// TwinCAT 3 PLC project H2AssemblyTesting
// ProgramVersion: 3.1.4026.17
// libraries:
//   Tc2_Standard, * (Beckhoff Automation GmbH)
//   Tc2_System, * (Beckhoff Automation GmbH)
//   Tc2_Utilities, * (Beckhoff Automation GmbH)
// project tree:
//   DUTs/ E_CompressionStages.TcDUT, E_ErrorState.TcDUT (not stored), E_InletToSystem.TcDUT (not stored), E_OutletNumber.TcDUT (not stored), E_TankBundleNumber.TcDUT (not stored), E_SolenoidState.TcDUT (not stored), ST_AnalogPressureTemp.TcDUT, ST_MatrixInputs.TcDUT, ST_Path.TcDUT (not stored), ST_SolenoidConfig.TcDUT
//   GVLs/ GVL_HMI.TcGVL, GVL_IO.TcGVL
//   / PlcTask.TcTTO (not stored)
//   POUs/ FB_Device.TcPOU, FB_IO.TcPOU, FB_Matrix.TcPOU, FB_PressureTransducer.TcPOU, FB_Solenoid.TcPOU, MAIN.TcPOU
//   POUs/Interfaces/ I_Devices.TcIO
// real-time tasks:
//   TASK PlcTask: cycle T#10ms, priority 20, ADS port 350
// I/O:
//   DEVICE Node 05 (disabled), AmsNetId 192.168.1.166.2.1
//     Node 05S0 [EK1100 EtherCAT Coupler (2A E-Bus)]
//       Node 05S2 [EL3058 8Ch. Ana. Input 4-20mA]
//       Node 05S4 [EL3058 8Ch. Ana. Input 4-20mA]
//       Node 05S6 [EL3058 8Ch. Ana. Input 4-20mA]
//       Node 05S8 [EL3058 8Ch. Ana. Input 4-20mA]
//       Node 05S10 [EL3058 8Ch. Ana. Input 4-20mA]
//       Node 05S11 [EL1904, 4 Ch. Safety Input 24V, TwinSAFE]
//         modules: Module 1 (FSOES)
//   DEVICE Node 06 (disabled), AmsNetId 192.168.1.166.3.1
//     Node 06S0 [EK1100 EtherCAT Coupler (2A E-Bus)]
//       Node 06S2 [EL2024 4Ch. Dig. Output 24V, 2A]
//       Node 06S4 [EL2024 4Ch. Dig. Output 24V, 2A]
//       Node 06S6 [EL2024 4Ch. Dig. Output 24V, 2A]
//       Node 06S8 [EL2024 4Ch. Dig. Output 24V, 2A]
//       Node 06S10 [EL2024 4Ch. Dig. Output 24V, 2A]
//       Node 06S12 [EL2024 4Ch. Dig. Output 24V, 2A]
//       Node 06S14 [EL2024 4Ch. Dig. Output 24V, 2A]
//       Node 06S16 [EL2024 4Ch. Dig. Output 24V, 2A]
// variable links:
//   H2AssemblyTesting/H2AssemblyTesting Instance <-> Node 05/Node 05S0/Node 05S2
//     PlcTask Inputs/GVL_IO.aPressRaw[{1..8}] <-> AI Standard Channel {1..8}/Value  (8 links)
//   H2AssemblyTesting/H2AssemblyTesting Instance <-> Node 05/Node 05S0/Node 05S4
//     PlcTask Inputs/GVL_IO.aPressRaw[10] <-> AI Standard Channel 2/Value
//     PlcTask Inputs/GVL_IO.aPressRaw[11] <-> AI Standard Channel 3/Value
//     PlcTask Inputs/GVL_IO.aPressRaw[12] <-> AI Standard Channel 4/Value
//     PlcTask Inputs/GVL_IO.aPressRaw[13] <-> AI Standard Channel 5/Value
//     PlcTask Inputs/GVL_IO.aPressRaw[14] <-> AI Standard Channel 8/Value
//     PlcTask Inputs/GVL_IO.aPressRaw[15] <-> AI Standard Channel 6/Value
//     PlcTask Inputs/GVL_IO.aPressRaw[16] <-> AI Standard Channel 7/Value
//     PlcTask Inputs/GVL_IO.aPressRaw[9] <-> AI Standard Channel 1/Value
//   H2AssemblyTesting/H2AssemblyTesting Instance <-> Node 05/Node 05S0/Node 05S6
//     PlcTask Inputs/GVL_IO.aTempRaw[{1..8}] <-> AI Standard Channel {1..8}/Value  (8 links)
//   H2AssemblyTesting/H2AssemblyTesting Instance <-> Node 05/Node 05S0/Node 05S8
//     PlcTask Inputs/GVL_IO.aTempRaw[10] <-> AI Standard Channel 2/Value
//     PlcTask Inputs/GVL_IO.aTempRaw[11] <-> AI Standard Channel 3/Value
//     PlcTask Inputs/GVL_IO.aTempRaw[12] <-> AI Standard Channel 4/Value
//     PlcTask Inputs/GVL_IO.aTempRaw[13] <-> AI Standard Channel 5/Value
//     PlcTask Inputs/GVL_IO.aTempRaw[14] <-> AI Standard Channel 8/Value
//     PlcTask Inputs/GVL_IO.aTempRaw[15] <-> AI Standard Channel 6/Value
//     PlcTask Inputs/GVL_IO.aTempRaw[16] <-> AI Standard Channel 7/Value
//     PlcTask Inputs/GVL_IO.aTempRaw[9] <-> AI Standard Channel 1/Value
//   H2AssemblyTesting/H2AssemblyTesting Instance <-> Node 06/Node 06S0/Node 06S10
//     PlcTask Outputs/GVL_IO.aFillMatrixValveCmds[{1..4},1] <-> Channel {1..4}/Output  (4 links)
//   H2AssemblyTesting/H2AssemblyTesting Instance <-> Node 06/Node 06S0/Node 06S12
//     PlcTask Outputs/GVL_IO.aDispenseMatrixValveCmds[{1..4},3] <-> Channel {1..4}/Output  (4 links)
//   H2AssemblyTesting/H2AssemblyTesting Instance <-> Node 06/Node 06S0/Node 06S14
//     PlcTask Outputs/GVL_IO.aDispenseMatrixValveCmds[{1..4},2] <-> Channel {1..4}/Output  (4 links)
//   H2AssemblyTesting/H2AssemblyTesting Instance <-> Node 06/Node 06S0/Node 06S16
//     PlcTask Outputs/GVL_IO.aDispenseMatrixValveCmds[{1..4},1] <-> Channel {1..4}/Output  (4 links)
//   H2AssemblyTesting/H2AssemblyTesting Instance <-> Node 06/Node 06S0/Node 06S2
//     PlcTask Outputs/GVL_IO.aInletMAtrixValveCmds[2,1] <-> Channel 1/Output
//     PlcTask Outputs/GVL_IO.aInletMAtrixValveCmds[2,2] <-> Channel 2/Output
//     PlcTask Outputs/GVL_IO.aInletMAtrixValveCmds[2,3] <-> Channel 3/Output
//   H2AssemblyTesting/H2AssemblyTesting Instance <-> Node 06/Node 06S0/Node 06S4
//     PlcTask Outputs/GVL_IO.aInletMAtrixValveCmds[1,1] <-> Channel 1/Output
//     PlcTask Outputs/GVL_IO.aInletMAtrixValveCmds[1,2] <-> Channel 2/Output
//     PlcTask Outputs/GVL_IO.aInletMAtrixValveCmds[1,3] <-> Channel 3/Output
//   H2AssemblyTesting/H2AssemblyTesting Instance <-> Node 06/Node 06S0/Node 06S6
//     PlcTask Outputs/GVL_IO.aFillMatrixValveCmds[{1..4},3] <-> Channel {1..4}/Output  (4 links)
//   H2AssemblyTesting/H2AssemblyTesting Instance <-> Node 06/Node 06S0/Node 06S8
//     PlcTask Outputs/GVL_IO.aFillMatrixValveCmds[{1..4},2] <-> Channel {1..4}/Output  (4 links)

// ---- DUTs/E_CompressionStages.TcDUT
{attribute 'strict'}
//Pathing Enum
TYPE E_CompressionStages :
(
	Bypass_Line:=1,
    Second_Stage_Compression:=2,
    First_Stage_Compression:=3
)USINT;
END_TYPE

// ---- DUTs/ST_AnalogPressureTemp.TcDUT
TYPE ST_AnalogPressureTemp :
	//Config struct for pressure/temp sensors
STRUCT
	rWarninglevel: LREAL;
	rErrorLevel: LREAL;
	rPressureMaxSP:LREAL;
	rPressureMinSP:LREAL;
	rTemperatureMaxSP:LREAL;
	rTemperatureMinSP:LREAL;
	nRawMax:INT;
	nRawMin:INT;
END_STRUCT
END_TYPE

// ---- DUTs/ST_MatrixInputs.TcDUT
TYPE ST_MatrixInputs :
STRUCT
	aManualValveSelection: ARRAY [1..GVL_HMI.cMaxRows,1..GVL_HMI.cMaxCols] OF BOOL;
	bTurnOnMatrix:BOOL;
	bResetMatrix:BOOL;
	bTurnOnPathing:BOOL;
	bActuatePath:BOOL;
	aStateofValves: ARRAY[1..GVL_HMI.cMaxRows,1..GVL_HMI.cMaxCols] OF E_SolenoidState;
END_STRUCT
END_TYPE

// ---- DUTs/ST_SolenoidConfig.TcDUT
TYPE ST_SolenoidConfig :
STRUCT
	NormallyOpen:BOOL; //True if valve to be configured as Normally open
    bOpen:BOOL; //True if valve should be opened
END_STRUCT
END_TYPE

// ---- GVLs/GVL_HMI.TcGVL
{attribute 'qualified_only'}
VAR_GLOBAL
	//Variables for the dispensing matrix
	eDispStartOfPath: E_TankBundleNumber;
	eDispEndOfPath:E_OutletNumber;
	//Variables for the inlet matrix
	eInletStartOfPath: E_InletToSystem;
	eInletEndOfPath:E_CompressionStages;
	//Variables for the Filling Matri
	eFillStartOfPath: E_TankBundleNumber;
	eFillEndOfPath:E_CompressionStages;
	//Input Structs for HMI to valve matrices
	stDispHMI:ST_MatrixInputs;
	stInletHMI : ST_MatrixInputs;
    stFillHMI  : ST_MatrixInputs;
	//Variable reset Sensors
	bResetSensors:BOOL;
	//Sensor Error states to display on HMI
	aSensorErrors :  ARRAY[1..GVL_IO.cNumofPT] OF E_ErrorState;
	//Sensor Engineering values
	aPV:  ARRAY[1..GVL_IO.cNumofPT] OF REAL;
	aTV:  ARRAY[1..GVL_IO.cNumofPT] OF REAL;
	//Overall Valve Reset
	bResetAllValves:BOOL;
	
END_VAR
VAR_GLOBAL CONSTANT
	//Set max matrix size at compile time
	cMaxRows:INT:=4;
	cMaxCols:INT:=3;
	cInletRows:INT:=2;
	cInletCols:INT:=3;
    cWarninglevel:LREAL:=500;
    cErrorLevel:LREAL:=525;
    cPressureMinSP:LREAL:=0;
    cPressureMaxSP:LREAL:=1000;
    cTemperatureMinSP:LREAL:=-40;
    cTemperatureMaxSP:LREAL:=125;
    cRawMin:	INT:=0;
    cRawMax:	INT:=32767;
END_VAR

// ---- GVLs/GVL_IO.TcGVL
{attribute 'qualified_only'}
VAR_GLOBAL CONSTANT
	cNumofPT:USINT:=16;
	cNumofMatrices:USINT:=3;
sPTTags : ARRAY[1..cNumofPT] OF T_MaxString := [
        'PT-301-A-II',
        'PT-302-A-II',
        'PT-350-A-II',
        'PT-351-A-II',
        'PT-352-A-II',
        'PT-353-A-II',
        'PT-354-A-II',
        'PT-355-A-II',
        'PT-356-A-II',
        'PT-357-A-II',
        'PT-358-A-II',
        'PT-359-A-II',
        'PT-360-A-II',
        'PT-365-A-II',
        'PT-361-A-II',
        'PT-363-A-II'
    ];
END_VAR
VAR_GLOBAL
	//Sensor Inputs
	aPressRaw AT %I*: ARRAY[1..cNumofPT] OF INT;
    aTempRaw AT %I* : ARRAY[1..cNumofPT]  OF INT;
	
	//Solenoid Outputs
	aInletMAtrixValveCmds AT %Q* : ARRAY [1..GVL_HMI.cInletRows,1..GVL_HMI.cInletCols] OF BOOL;
	aFillMatrixValveCmds AT %Q*: ARRAY [1..GVL_HMI.cMaxRows,1..GVL_HMI.cMaxCols] OF BOOL;
	aDispenseMatrixValveCmds AT %Q*: ARRAY [1..GVL_HMI.cMaxRows,1..GVL_HMI.cMaxCols] OF BOOL;
END_VAR

// ---- POUs/Interfaces/I_Devices.TcIO
INTERFACE I_Devices

METHOD M_CyclicLogic : HRESULT
END_METHOD

END_INTERFACE

// ---- POUs/FB_Device.TcPOU
FUNCTION_BLOCK PUBLIC FB_Device IMPLEMENTS I_Devices
//Base class for matrix, solenoid and PTTransducer classes
VAR_INPUT
	bDeviceEnable:BOOL; //Make the device Active
	bDeviceReset:BOOL;//Reset Error state
END_VAR
VAR_OUTPUT
    bError        : BOOL;   // True if in error
	bWarning :BOOL; //True if warning applicable
    eDeviceState  : E_ErrorState; // Summary device state
END_VAR
VAR
	hr : HRESULT;
	fbTrig:R_TRIG;
END_VAR

METHOD PUBLIC M_CyclicLogic : HRESULT
//  Check enable state
IF NOT bDeviceEnable THEN
	eDeviceState:=E_ErrorState.Disabled;
	M_CyclicLogic := S_Pending;
	RETURN;
END_IF

// Check reset 
fbTrig(CLK:=bDeviceReset);
IF fbTrig.Q THEN
	bError:=FALSE;
	bWarning:=FALSE;
	eDeviceState:=E_ErrorState.Healthy;
END_IF

// Handle state logic
IF bError THEN
	eDeviceState:=E_ErrorState.Alarm;
	M_CyclicLogic := E_FAIL;
ELSIF bWarning THEN
        eDeviceState:=E_ErrorState.Warning;	
		M_CyclicLogic := S_Pending;
ELSE 
		eDeviceState:=E_ErrorState.Healthy;
		M_CyclicLogic := S_OK;
END_IF
END_METHOD

END_FUNCTION_BLOCK

// ---- POUs/FB_IO.TcPOU
FUNCTION_BLOCK PUBLIC FB_IO
VAR_INPUT
	PTTT: REFERENCE TO ARRAY [1.. GVL_IO.cNumofPT] OF FB_PressureTransducer;
END_VAR
VAR
	inlet:FB_matrix;
	fill:FB_matrix;
	dispense:FB_matrix;
	nsensorNumber:INT;
	rows:INT;
	cols:INT;
	aInletMAtrixValveCmds: INT;
END_VAR

M_PTTTransducers();
M_Solenoids();

PROPERTY DispenseMatrix : FB_matrix
SET
dispense := DispenseMatrix;
END_SET
END_PROPERTY

PROPERTY FillMatrix : FB_matrix
SET
fill := FillMatrix;
END_SET
END_PROPERTY

PROPERTY InletMatrix : FB_matrix
SET
inlet := InletMatrix;
END_SET
END_PROPERTY

METHOD M_PTTTransducers
FOR nsensorNumber:=1 TO GVL_IO.cNumofPT DO		
    PTTT[nsensorNumber].RawPressure := GVL_IO.aPressRaw[nsensorNumber];
    PTTT[nsensorNumber].RawTemperature := GVL_IO.aTempRaw[nsensorNumber];
END_FOR
END_METHOD

METHOD M_Solenoids
//Update IO for valve commands
FOR rows:=1 TO GVL_HMI.cInletRows DO
	FOR cols:=1 TO GVL_HMI.cInletCols DO
	    GVL_IO.aInletMAtrixValveCmds[rows,cols]:= inlet.aValveCommands[rows,cols];
	END_FOR
END_FOR
FOR rows:=1 TO GVL_HMI.cMaxRows DO
	FOR cols:=1 TO GVL_HMI.cMaxCols DO
	    GVL_IO.aFillMatrixValveCmds[rows,cols]:= fill.aValveCommands[rows,cols];
		GVL_IO.aDispenseMatrixValveCmds[rows,cols]:= Dispense.aValveCommands[rows,cols];
	END_FOR
END_FOR
END_METHOD

END_FUNCTION_BLOCK

// ---- POUs/FB_PressureTransducer.TcPOU
FUNCTION_BLOCK FB_PressureTransducer EXTENDS FB_Device 
VAR
	nSensorPressure: INT; //Pressure analog input
	nSensorTemperature: INT;//Temperature analog input 
	st_AnalogPressureTempdata:ST_AnalogPressureTemp;//Configuration struct 
	sTag : T_MaxString;
	rEngPressure:REAL;//Pressure in BAR.
	rEngTemperature:REAL;//Temperature in Degrees C.
END_VAR

PROPERTY EngPressure : LREAL
GET
EngPressure := rEngPressure;
END_GET
END_PROPERTY

PROPERTY EngTemperature : LREAL
GET
EngTemperature := rEngTemperature;
END_GET
END_PROPERTY

METHOD M_CyclicLogic :HRESULT
VAR
	rNormPressure:REAL;
	rNormTemperature:REAL;
END_VAR
//Call M_CyclicLogic from FB_Device 
hr:=SUPER^.M_CyclicLogic();
IF bDeviceEnable THEN
	//Normalise the analog inputs 
   rNormPressure    := (INT_TO_REAL(nSensorPressure)    - INT_TO_REAL(st_AnalogPressureTempdata.nRawMin)) / (INT_TO_REAL(st_AnalogPressureTempdata.nRawMax) - INT_TO_REAL(st_AnalogPressureTempdata.nRawMin));
   rNormTemperature := (INT_TO_REAL(nSensorTemperature) - INT_TO_REAL(st_AnalogPressureTempdata.nRawMin)) / (INT_TO_REAL(st_AnalogPressureTempdata.nRawMax) - INT_TO_REAL(st_AnalogPressureTempdata.nRawMin));
   
   //Scale analog inputs to the Engineering process values, using config struct parameters
   rEngPressure:=st_AnalogPressureTempdata.rPressureMinSP + rNormPressure * (st_AnalogPressureTempdata.rPressureMaxSP - st_AnalogPressureTempdata.rPressureMinSP);
   rEngTemperature:=st_AnalogPressureTempdata.rTemperatureMinSP + rNormTemperature * (st_AnalogPressureTempdata.rTemperatureMaxSP - st_AnalogPressureTempdata.rTemperatureMinSP);
END_IF

//Evaluate pressure state 
M_PressureState();
END_METHOD

METHOD M_Init 
VAR_INPUT
    sTag  : T_MaxString;
END_VAR
VAR
	stCfg : ST_AnalogPressureTemp;
END_VAR
//COnfigure the config struct parameters
stCfg.rWarninglevel := GVL_HMI.cWarninglevel;
stCfg.rErrorLevel := GVL_HMI.cErrorLevel;
stCfg.rPressureMinSP := GVL_HMI.cPressureMinSP;
stCfg.rPressureMaxSP := GVL_HMI.cPressureMaxSP;
stCfg.rTemperatureMinSP := GVL_HMI.cTemperatureMinSP;
stCfg.rTemperatureMaxSP := GVL_HMI.cTemperatureMaxSP;
stCfg.nRawMin := GVL_HMI.cRawMin;
stCfg.nRawMax := GVL_HMI.cRawMax;

st_AnalogPressureTempdata:=stCfg;
bDeviceEnable:=TRUE;
THIS^.sTag:=sTag;
END_METHOD

METHOD M_PressureState
//Evaluate pressure value against warning and error values.
IF (rEngPressure > st_AnalogPressureTempdata.rWarninglevel) AND (rEngPressure < st_AnalogPressureTempdata.rErrorLevel) THEN
	bWarning:=TRUE;
ELSIF rEngPressure > st_AnalogPressureTempdata.rErrorLevel THEN
	bError:=TRUE;
ELSE 
	bWarning:=FALSE;
END_IF
END_METHOD

METHOD M_UpdateToHMI 
VAR_OUTPUT
	PV : REAL;
	TV : REAL;
	State : E_ErrorState;
END_VAR
PV := EngPressure;
TV := EngTemperature;
State := SensorState;
END_METHOD

PROPERTY RawPressure :  INT
SET
nSensorPressure := RawPressure;
END_SET
END_PROPERTY

PROPERTY RawTemperature :  INT
SET
nSensorTemperature := RawTemperature;
END_SET
END_PROPERTY

PROPERTY SensorState : E_ErrorState
GET
SensorState := eDeviceState;
END_GET
END_PROPERTY

END_FUNCTION_BLOCK

// ---- POUs/FB_Matrix.TcPOU
FUNCTION_BLOCK FB_Matrix EXTENDS FB_Device 
VAR
	st_path : ST_Path;//INT struct to contain int value of path enums
	bSetCurrentPath:BOOL;//Bool to actuate the selected path 
	bPathingOn:BOOL;//BOOL to enable the path selection mode 
	aValves:ARRAY [1..GVL_HMI.cMaxRows,1..GVL_HMI.cMaxCols] OF FB_Solenoid;//Instantiating Solenoid valves, max array size, can contain smaller arrays
	iRows:INT;//Row variable for FOR loops to use
	iColumns:INT;//Col variable for FOR loops to use
	bOverallEnable:BOOL;//Internal variable used to assign device state to all instantiated solenoid valves
	nRowSize:INT;//Matrix row size 
	nColSize:INT;//Matrix Column size
	aConfig:ARRAY[1..GVL_HMI.cMaxRows,1..GVL_HMI.cMaxCols] OF ST_SolenoidConfig;//Matrix config
	aValveStates : ARRAY [1..GVL_HMI.cMaxRows,1..GVL_HMI.cMaxCols] OF E_SolenoidState;//State of valves
	aLastCmdTime : ARRAY[1..GVL_HMI.cMaxRows, 1..GVL_HMI.cMaxCols] OF DT;
	aPrevOpen    : ARRAY[1..GVL_HMI.cMaxRows, 1..GVL_HMI.cMaxCols] OF BOOL;
END_VAR
VAR_OUTPUT
	aValveCommands:ARRAY [1..GVL_HMI.cMaxRows,1..GVL_HMI.cMaxCols] OF BOOL;
END_VAR

METHOD M_CyclicLogic : HRESULT
//Call FB_Device M_Cyclic Logic
hr:=SUPER^.M_CyclicLogic();
M_EnableResetLogic();
IF bDeviceEnable AND bPathingON THEN
	
	M_DispensePathing();
	
END_IF

M_SafteyLogic();

   FOR iRows := 1 TO nRowSize DO
       FOR iColumns := 1 TO nColSize DO
		   
           aValves[iRows, iColumns](
              bDeviceEnable:=bOverallEnable,
		      bNormallyOpen:=aConfig[iRows,iColumns].NormallyOpen,
              bCmdOpen:=aConfig[iRows,iColumns].bOpen,
              bCoilEnergiseState=>aValveCommands[iRows,iColumns]);
			  
			  aValveStates[iRows, iColumns]:=aValves[iRows, iColumns].eSolenoidState;
              aPrevOpen[iRows, iColumns] := aConfig[iRows, iColumns].bOpen;
       END_FOR
   END_FOR
END_METHOD

METHOD PRIVATE M_DispensePathing 
VAR
	nRowToOpen: INT :=(st_path.startPath);
	nColToOpen: INT :=(st_path.endPath);
END_VAR
IF bSetCurrentPath THEN
	// Clear all valves in active area 
    FOR iRows := 1 TO nRowSize DO
        FOR iColumns := 1 TO nColSize DO
            aConfig[iRows, iColumns].bOpen := FALSE;
        END_FOR
    END_FOR
   aConfig[nRowToOpen,nColToOpen].bOpen:=TRUE;
END_IF
END_METHOD

METHOD PRIVATE M_EnableResetLogic
//Set up variables and logic to reset and enable valve FB's created by FB_Matrix
bOverallEnable:=bDeviceEnable;
IF bDeviceReset THEN
    FOR iRows := 1 TO nRowSize DO
       FOR iColumns := 1 TO nColSize DO
           aValves[iRows, iColumns](bDeviceReset:=fbTrig.Q);
		   aConfig[iRows,iColumns].bOpen:=FALSE;
       END_FOR
    END_FOR
END_IF
END_METHOD

METHOD M_Init : HRESULT
VAR_INPUT
	nRows:INT;//Matrix row size 
	nCols:INT;//Matrix Column size
END_VAR
VAR
    x:INT;
	y:INT;
END_VAR
//Set size of matrix	
IF nRows > GVL_HMI.cMaxRows OR nCols > GVL_HMI.cMaxCols THEN
	M_Init := E_FAIL;
	RETURN;
END_IF
    nRowSize:=nRows;
	nColSize:=nCols;
//Initialise aConfig as NC and valves closed
FOR x:= 1 TO nRowSize DO
    FOR y := 1 TO nColSize DO
        aConfig[x, y].bOpen        := FALSE;
        aConfig[x, y].NormallyOpen := FALSE;
    END_FOR
END_FOR
M_Init:= S_OK;
END_METHOD

METHOD PRIVATE M_ManualControl 
VAR_INPUT
		stHMI:ST_MatrixInputs;
END_VAR
FOR iRows := 1 TO nRowSize DO
    FOR iColumns := 1 TO nColSize DO
        aConfig[iRows, iColumns].bOpen := stHMI.aManualValveSelection[iRows, iColumns];
    END_FOR
END_FOR
END_METHOD

METHOD PRIVATE M_ResetValves 
VAR_IN_OUT
	stHMI:ST_MatrixInputs;
END_VAR
IF bDeviceReset THEN
    FOR iRows := 1 TO nRowSize DO
        FOR iColumns := 1 TO nColSize DO
            stHMI.aManualValveSelection[iRows, iColumns] := FALSE;
        END_FOR
    END_FOR
END_IF
END_METHOD

METHOD PRIVATE M_SafteyLogic 
VAR
    a, b, winnerA, winnerB: INT; 
END_VAR
M_UpdateTime();
// Row pass
FOR a := 1 TO nRowSize DO
    winnerB := 0;
    // Pick the newest-open valve in this row
    FOR b := 1 TO nColSize DO
        IF aConfig[a, b].bOpen THEN
            IF winnerB = 0 THEN
                winnerB := b;
            ELSE
                // Compare timestamps
                IF aLastCmdTime[a, b] >= aLastCmdTime[a, winnerB] THEN
                    winnerB := b;
                END_IF
            END_IF
        END_IF
    END_FOR

    // Close losers
    IF winnerB <> 0 THEN
        FOR b := 1 TO nColSize DO
            IF b <> winnerB THEN
                aConfig[a, b].bOpen := FALSE;
            END_IF
        END_FOR
    END_IF
END_FOR

// Columns
FOR b := 1 TO nColSize DO
    winnerA := 0;
    FOR a := 1 TO nRowSize DO
        IF aConfig[a, b].bOpen THEN

            IF winnerA = 0 THEN
                winnerA := a;
            ELSE
                IF aLastCmdTime[a, b] >= aLastCmdTime[winnerA, b] THEN
                    winnerA := a;
                END_IF
            END_IF
        END_IF
    END_FOR

    // Close losers
    IF winnerA <> 0 THEN
        FOR a := 1 TO nRowSize DO
            IF a <> winnerA THEN
                aConfig[a, b].bOpen := FALSE;
            END_IF
        END_FOR
    END_IF
END_FOR
END_METHOD

METHOD PUBLIC M_UpdateFromHMI : BOOL
VAR_IN_OUT
	stHMI:ST_MatrixInputs;
END_VAR
VAR_INPUT
	nStartOfPath : INT; 
    nEndOfPath   : INT;
END_VAR
bDeviceEnable := stHMI.bTurnOnMatrix;
bDeviceReset := stHMI.bResetMatrix OR GVL_HMI.bResetAllValves;
bPathingOn := stHMI.bTurnOnPathing;
bSetCurrentPath := stHMI.bActuatePath;
st_path.startPath := nStartOfPath;
st_path.endPath := nEndOfPath;


M_ResetValves(stHMI := stHMI);

IF bPathingOn THEN;
	RETURN;
END_IF

M_ManualControl(stHMI := stHMI);
END_METHOD

METHOD PRIVATE M_UpdateTime 
VAR
	 // System time internals
    fbSystemTime : GETSYSTEMTIME;
    stFileTime   : T_FILETIME;
    dtNow        : DT;  
	a , b : INT;
END_VAR
// Read system time 
fbSystemTime(
    timeLoDW => stFileTime.dwLowDateTime,
    timeHiDW => stFileTime.dwHighDateTime
);

// Convert to DT Type
dtNow := FILETIME_TO_DT(stFileTime);

FOR a := 1 TO nRowSize DO
    FOR b := 1 TO nColSize DO

        IF aConfig[a, b].bOpen AND NOT aPrevOpen[a, b] THEN
            aLastCmdTime[a, b] := dtNow;   
        END_IF
		
    END_FOR
END_FOR
END_METHOD

METHOD PUBLIC M_UpdateToHMI : BOOL
VAR_IN_OUT
    stHMI : ST_MatrixInputs;
END_VAR
FOR iRows := 1 TO GVL_HMI.cmaxRows DO
    FOR iColumns := 1 TO GVL_HMI.cMaxCols DO
        stHMI.aManualValveSelection[iRows,iColumns]:=aConfig[iRows,iColumns].bOpen;
    END_FOR
END_FOR
FOR iRows := 1 TO nRowSize DO
    FOR iColumns := 1 TO nColSize DO
        stHMI.aStateOfValves[iRows, iColumns] := aValveStates[iRows, iColumns];
    END_FOR
END_FOR
END_METHOD

END_FUNCTION_BLOCK

// ---- POUs/FB_Solenoid.TcPOU
FUNCTION_BLOCK FB_Solenoid EXTENDS FB_Device
VAR_INPUT
	bNormallyOpen:BOOL;//True if Valve is Normally Open
	bCmdOpen:BOOL;// True if Valve should be opened
END_VAR
VAR
	bTheoreticallyOpen:BOOL;//Internal variable to control state of the valve, true when valve is open
END_VAR
VAR_OUTPUT
	bCoilEnergiseState:BOOL;//Signal sent to coil to energise
	eSolenoidState: E_SolenoidState;//If coil is not energised in reality
END_VAR

//Call method open or close depending on command to valve
IF bCmdOpen THEN
	M_Open();
ELSE
    M_Close();
END_IF

METHOD M_CheckState
//Return the state enum of the valve 
IF bTheoreticallyOpen THEN
	eSolenoidState := E_SolenoidState.Open;
ELSE
	eSolenoidState := E_SolenoidState.Closed;
END_IF
END_METHOD

METHOD PUBLIC M_Close
//Call base M_Cyclic logic from FB_Device
hr:=SUPER^.M_CyclicLogic();
//Close the valve if the device is enabled
IF bDeviceEnable THEN
	IF bNormallyOpen THEN
		bCoilEnergiseState := TRUE;
		bTheoreticallyOpen := FALSE;
	ELSE
		bCoilEnergiseState := FALSE;
		bTheoreticallyOpen := bNormallyOpen;
	END_IF
ELSE
	bCoilEnergiseState := FALSE;
	bTheoreticallyOpen := bNormallyOpen;
END_IF
M_CheckState();
END_METHOD

METHOD PUBLIC M_Open
////Call base M_Cyclic logic from FB_Device
hr:=SUPER^.M_CyclicLogic();
//Open the valve if the device is enabled
IF bDeviceEnable THEN
	IF NOT bNormallyOpen THEN
		bCoilEnergiseState := TRUE;
		bTheoreticallyOpen := TRUE;
	ELSE
		bCoilEnergiseState := FALSE;
		bTheoreticallyOpen := bNormallyOpen;
	END_IF
ELSE
	bCoilEnergiseState := FALSE;
	bTheoreticallyOpen := bNormallyOpen;
END_IF
M_Checkstate();
END_METHOD

END_FUNCTION_BLOCK

// ---- POUs/MAIN.TcPOU
PROGRAM MAIN
VAR
	//Matrix instances
	fbDispenseMatrix : FB_Matrix;
	fbInletMatrix : FB_Matrix;
	fbFillMatrix : FB_Matrix;

	//Instance of fbIO for IO updates
	fbIO : FB_IO;
	
	//Pressure Transducers
	aPT : ARRAY [1.. GVL_IO.cNumofPT] OF FB_PressureTransducer;
	
	//Devices interface
	Devices : ARRAY[1..GVL_IO.cNumofMatrices+GVL_IO.cNumofPT] OF I_Devices;
	
	//Initialising Boolean 
	bInitialise : BOOL := TRUE;
	
	idx : USINT;
	
	hr : HRESULT := S_PENDING;
END_VAR

//Run Initialise Method once on first cycle
IF bInitialise THEN
	hr := M_Initalize();
	RETURN;
END_IF

//Update IO
M_UpdateIO(PTTT:=aPT);

//Update From HMI
M_UpdateFromHMI();	

//Calling Cyclic
M_CyclicLogic();

//Update HMI
M_UpdateToHMI();

METHOD M_CyclicLogic
FOR idx := 1 TO GVL_IO.cNumofMatrices+GVL_IO.cNumofPT DO
    Devices[idx].M_CyclicLogic();
END_FOR
END_METHOD

METHOD PUBLIC M_Initalize : HRESULT
VAR
idx : INT;
// Config Parameter Struct 
stAnalogCfg : ST_AnalogPressureTemp;
hresult: ARRAY[1..GVL_IO.cNumofMatrices] OF HRESULT;
END_VAR

//Assign Devices into Interface array
Devices[1] := fbDispenseMatrix;
Devices[2] := fbInletMatrix;
Devices[3] := fbFillMatrix;
	
FOR idx := 1 TO GVL_IO.cNumofPT DO
    Devices[GVL_IO.cNumofMatrices + idx] := aPT[idx];
END_FOR
	
//Initialise the pressure sensors
FOR idx:=1 TO GVL_IO.cNumofPT DO
    aPT[idx].M_Init(sTag:=GVL_IO.sPTTags[idx]);
END_FOR

//Initialise matrices 
hresult[1] := fbInletMatrix.M_Init(nRows:=GVL_HMI.cInletRows,nCols:=GVL_HMI.cInletCols);
hresult[2] :=fbDispenseMatrix.M_Init(nRows:=GVL_HMI.cMaxRows,nCols:=GVL_HMI.cMaxCols);
hResult[3] := fbFillMatrix.M_Init(nRows:=GVL_HMI.cMaxRows,nCols:=GVL_HMI.cMaxCols);

//Logic to check if matrices fail to initialise
FOR idx:= 1 TO GVL_IO.cNumofMatrices DO
	IF hresult[idx] = E_FAIL THEN
		M_Initalize:= E_FAIL;
		RETURN;
	END_IF
END_FOR

//Initialised succesfully
bInitialise:=FALSE;
M_Initalize := S_OK;
END_METHOD

METHOD M_UpdateFromHMI
//Update each matrix using its update method
fbDispenseMAtrix.M_UpdateFromHMI(stHMI:=GVL_HMI.stDispHMI,
	                             nStartOfPath:=GVL_HMI.eDispStartOfPath,
								 nEndOfPath:=GVL_HMI.eDispEndOfPath);
								 
fbFillMatrix.M_UpdateFromHMI(stHMI:=GVL_HMI.stFillHMI,
	                             nStartOfPath:=GVL_HMI.eFillStartOfPath,
								 nEndOfPath:=GVL_HMI.eFillEndOfPath);
								 
fbInletMatrix.M_UpdateFromHMI(stHMI:=GVL_HMI.stInletHMI,
	                             nStartOfPath:=GVL_HMI.eInletStartOfPath,
								 nEndOfPath:=GVL_HMI.eInletEndOfPath);
END_METHOD

METHOD M_UpdateIO 
VAR_INPUT
	PTTT: REFERENCE TO ARRAY [1.. GVL_IO.cNumofPT] OF FB_PressureTransducer;
END_VAR
fbIO.DispenseMatrix:=fbDispenseMatrix;
fbIO.FillMatrix:=fbFillMatrix;
fbIO.InletMatrix:=fbInletMatrix;
fbIO(PTTT:=aPT);
END_METHOD

METHOD M_UpdateToHMI
VAR
	idx : INT;
END_VAR
fbDispenseMatrix.M_UpdateToHMI(stHMI:=GVL_HMI.stDispHMI);
fbFillMatrix.M_UpdateToHMI(stHMI:=GVL_HMI.stFillHMI);
fbInletMatrix.M_UpdateToHMI(stHMI:=GVL_HMI.stInletHMI);
FOR idx:=1 TO GVL_IO.cNumofPT DO
	aPT[idx].M_UpdateToHMI(PV=>GVL_HMI.aPV[idx],
		                   TV=>GVL_HMI.aTV[idx],
						   State=>GVL_HMI.aSensorErrors[idx]);
END_FOR
END_METHOD

END_PROGRAM
